TEXTLIST txtLstMotorEnableMode
  0 = 'Off'
  1 = 'Both Dir'
  2 = 'Only CW'
  3 = 'Only CCW'
   = ''
END_TEXTLIST

(* stored: Version 1.1.0.1, ProductVersion 3.1.4019.2
   TextList txtLstMotorEnableMode: Id {c5b1ce44-5d92-4bba-8049-3124899cc5e8} *)
